{attribute 'GeneratedUsingTerminal: EL6201-0000-0017'}
{attribute addProperty BoxType "EL6201-0000-0017"}
{attribute addProperty Id "Slave_12A_DO0BOOL1Slave_12A_DO1BOOL1Slave_12A_DO2BOOL1Slave_12A_DO3BOOL1Slave_12B_DO0BOOL1Slave_12B_DO1BOOL1Slave_12B_DO2BOOL1Slave_12B_DO3BOOL1"}
{attribute addProperty CRC "2886380969"}
{attribute addProperty Size "8"}
TYPE Slave_12_Outputs_AC0AADA9 :
STRUCT
	{attribute addProperty Name "Slave_12A_DO0"}
	Slave_12A_DO0 : BOOL;
	{attribute addProperty Name "Slave_12A_DO1"}
	Slave_12A_DO1 : BOOL;
	{attribute addProperty Name "Slave_12A_DO2"}
	Slave_12A_DO2 : BOOL;
	{attribute addProperty Name "Slave_12A_DO3"}
	Slave_12A_DO3 : BOOL;
	{attribute addProperty Name "Slave_12B_DO0"}
	Slave_12B_DO0 : BOOL;
	{attribute addProperty Name "Slave_12B_DO1"}
	Slave_12B_DO1 : BOOL;
	{attribute addProperty Name "Slave_12B_DO2"}
	Slave_12B_DO2 : BOOL;
	{attribute addProperty Name "Slave_12B_DO3"}
	Slave_12B_DO3 : BOOL;
END_STRUCT
END_TYPE

(* stored: Version 1.2.0.0, ProductVersion 3.1.4024.9
   DUT Slave_12_Outputs_AC0AADA9: Id {054d289e-db68-481a-8cf2-73b62e82cead} *)
